(* CODESYS project TUGAS AKHIR.project

Project tree, tasks and I/O mapping:
  Device : CODESYS Control Win V3, 3S - Smart Software Solutions GmbH, version 3.5.3.0
    application Application
      libraries: Standard, 3.5.2.0 (System)
      task MainTask (cyclic, interval t#20ms, priority 1) calls PLC_PRG
      task VISU_TASK (cyclic, interval 100 ms, priority 30) calls VisuElems.Visu_Prg
      program PLC_PRG [LD]
      visualisation Visualization
  CODESYS_Control_Win_V3 : CODESYS Control Win V3, 3S - Smart Software Solutions GmbH, version 3.5.3.0
    application Application
  text list GlobalTextList
*)

// Device/Application/PLC_PRG
PROGRAM PLC_PRG
VAR
	sensor1: BOOL;
	sensor2: BOOL;
	sensor3: BOOL;
	limitswicth1:BOOL;
	limitswicth2:BOOL;
	limitswicth3:BOOL;
	motor1maju:BOOL;
	motor2maju:BOOL;
	motor3maju:BOOL;
    motor1mundur:BOOL;
	motor2mundur:BOOL;
	motor3mundur:BOOL;
	t1: BOOL;
	t2: BOOL;
	t3: BOOL;
	tim1 : TON;
	tim2 : TON;
	tim3 : TON;
END_VAR

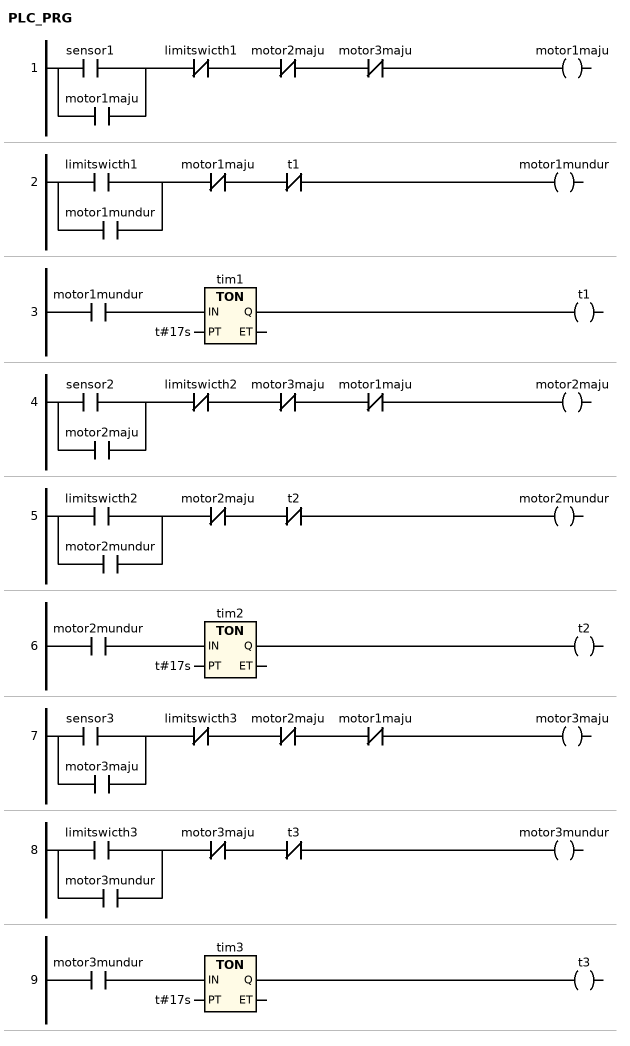
// NETWORK 1
motor1maju := (sensor1 OR motor1maju) AND NOT limitswicth1 AND NOT motor2maju AND NOT motor3maju;

// NETWORK 2
motor1mundur := (limitswicth1 OR motor1mundur) AND NOT motor1maju AND NOT t1;

// NETWORK 3
tim1(IN := motor1mundur, PT := t#17s); // TON
t1 := tim1.Q;

// NETWORK 4
motor2maju := (sensor2 OR motor2maju) AND NOT limitswicth2 AND NOT motor3maju AND NOT motor1maju;

// NETWORK 5
motor2mundur := (limitswicth2 OR motor2mundur) AND NOT motor2maju AND NOT t2;

// NETWORK 6
tim2(IN := motor2mundur, PT := t#17s); // TON
t2 := tim2.Q;

// NETWORK 7
motor3maju := (sensor3 OR motor3maju) AND NOT limitswicth3 AND NOT motor2maju AND NOT motor1maju;

// NETWORK 8
motor3mundur := (limitswicth3 OR motor3mundur) AND NOT motor3maju AND NOT t3;

// NETWORK 9
tim3(IN := motor3mundur, PT := t#17s); // TON
t3 := tim3.Q;

END_PROGRAM

// Device/Application/Visualization
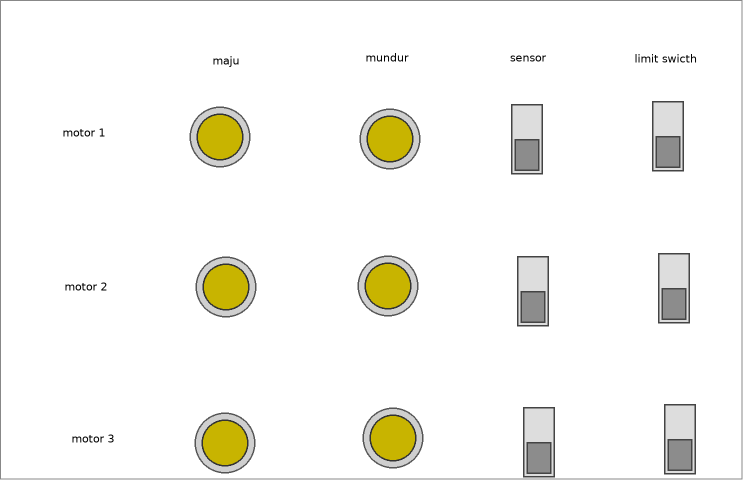
VISUALIZATION Visualization  // 743x480
    Lamp1 (185,102 70x70), variable: PLC_PRG.motor1maju, style: Lamp-Lamp1-Yellow
    Lamp1 (355,104 70x70), variable: PLC_PRG.motor1mundur, style: Lamp-Lamp1-Yellow
    Lamp1 (190,408 70x70), variable: PLC_PRG.motor3maju, style: Lamp-Lamp1-Yellow
    Lamp1 (358,403 70x70), variable: PLC_PRG.motor3mundur, style: Lamp-Lamp1-Yellow
    Lamp1 (191,252 70x70), variable: PLC_PRG.motor2maju, style: Lamp-Lamp1-Yellow
    Lamp1 (353,251 70x70), variable: PLC_PRG.motor2mundur, style: Lamp-Lamp1-Yellow
    Label (9,118 150x30), "motor 1"
    Label (11,272 150x30), "motor 2"
    Label (18,424 150x30), "motor 3"
    Label (151,46 150x30), "maju"
    Label (312,43 150x30), "mundur"
    DipSwitch (492,104 70x70), variable: PLC_PRG.sensor1, behaviour: TOGGLE, style: Switch-DipSwitch-Gray
    DipSwitch (498,256 70x70), variable: PLC_PRG.sensor2, behaviour: TOGGLE, style: Switch-DipSwitch-Gray
    DipSwitch (504,407 70x70), variable: PLC_PRG.sensor3, behaviour: TOGGLE, style: Switch-DipSwitch-Gray
    Label (453,43 150x30), "sensor"
    DipSwitch (633,101 70x70), variable: PLC_PRG.limitswicth1, behaviour: TOGGLE, style: Switch-DipSwitch-Gray
    DipSwitch (639,253 70x70), variable: PLC_PRG.limitswicth2, behaviour: TOGGLE, style: Switch-DipSwitch-Gray
    DipSwitch (645,404 70x70), variable: PLC_PRG.limitswicth3, behaviour: TOGGLE, style: Switch-DipSwitch-Gray
    Label (591,44 150x30), "limit swicth"
END_VISUALIZATION
